FUNCTION_BLOCK TcaStorage EXTENDS TcoCore.TcoComponent

VAR_INPUT
	ref : REFERENCE TO TcaStorageRef;
END_VAR

VAR	
	_Dock : BOOL;
	_Carrier : TcaCarrier(THIS^);
	_CarrierSensor : TcoDi(THIS^);	
	_CarrierPresent : BOOL;

	_Task : TcoCore.TcoTask(THIS^);	
	_cmd : eTcaStorageCmd;
	
	// Carrier Setting
	fbCarrierTemplate	: TcaCarrier(THIS^);	

END_VAR

IF NOT __ISVALIDREF(ref) THEN
	_Dock := FALSE;
ELSE
	_Dock := TRUE;
	_CarrierSensor(inoSignal := ref.Sensor);
END_IF


IF _Task.Done THEN
	_Task.Restore();
END_IF


IF _Task.Execute() THEN
	RETURN;
END_IF


CASE _cmd OF
	
	eTcaStorageCmd.FillCarrier:
		AddCarrier().FillWithWorkpieces_InitialStatus();
			
	eTcaStorageCmd.RemoveCarrier:
		RemoveCarrier();
	
	eTcaStorageCmd.EmptyCarrier:
		;
	
END_CASE
	

_Task.DoneWhen(TRUE);

METHOD AddCarrier : REFERENCE TO TcaCarrier
_CarrierPresent := TRUE;
_Carrier.Restore();
AddCarrier REF= _Carrier;
END_METHOD

PROPERTY CarrierPresent : BOOL
GET
CarrierPresent := _CarrierSensor.Signal;
END_GET
END_PROPERTY

METHOD RemoveCarrier : REFERENCE TO TcaCarrier
VAR
END_VAR
_CarrierPresent := FALSE;
_Carrier.Restore();
RemoveCarrier REF= _Carrier;
END_METHOD

(*~
	<docu>
		<summary>
			Restores this instance to the Ready state. Can be called explicitly or from within one of the restore mechanisms.	
		</summary>			
	</docu>	
~*)
METHOD Restore : TcoCore.ITcoRestorable
END_METHOD

(*~
	<docu>
		<summary>
		    Custom service (manual, maintenance) logic.
			This method must be implemented in derived class.
		</summary>			
	</docu>	
~*)
METHOD PROTECTED ServiceMode
_Carrier.Service();
END_METHOD

END_FUNCTION_BLOCK

(* stored: Version 1.1.0.1
   POU TcaStorage: Id {adbdc0ab-b9f5-4855-86de-ec4993fc6338}, SpecialFunc None
   Folder Operations: Id {0d9d7aea-b4a4-458e-b42d-8e40bf8aa761}
   Folder Properties: Id {601d726d-4565-4b3c-86fa-05ba78fa390f}
   Folder Tasks: Id {5ae2a9d4-1f46-4e18-bdf6-73c7fcb30846}
   Method AddCarrier: Id {615c98f7-b5f8-4b1e-9e24-1fa1c511ed65}
   Property CarrierPresent: Id {f89f5b0f-f321-451d-acf3-71e48130cfd0}
   Get Get: Id {5da2aca9-3120-46ce-9bc1-6e8430ccbb54}
   Method RemoveCarrier: Id {498c08c5-7e6c-491a-b470-1cb7bf5317e2}
   Method Restore: Id {55f00be3-3904-4111-ad40-1755c9e1a58b}
   Method ServiceMode: Id {c4d0b5e5-96b9-4510-8d72-a260e7c5a36a} *)
